Xinje XDPPro project, PLC1: XD3-48 (software 3.8.0 2025-09-09)

PROGRAM Ladder

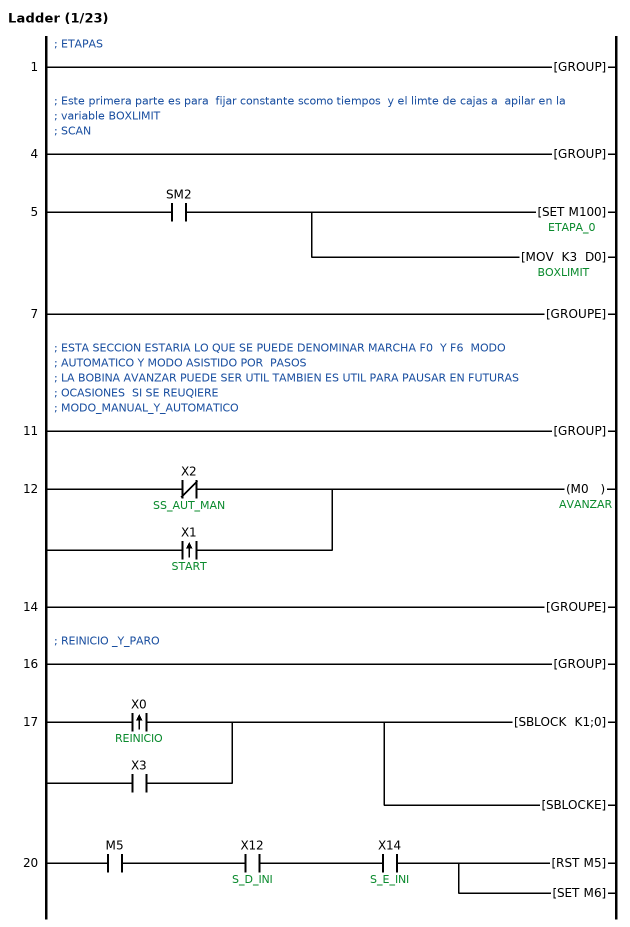
; ETAPAS
GROUP
; Este primera parte es para  fijar constante scomo tiempos  y el limte de cajas a  apilar en la variable BOXLIMIT
; SCAN
GROUP
LD     SM2
SET    M100	; ETAPA_0
MOV    K3 D0	; BOXLIMIT
GROUPE
; ESTA SECCION ESTARIA LO QUE SE PUEDE DENOMINAR MARCHA F0  Y F6  MODO AUTOMATICO Y MODO ASISTIDO POR  PASOS
; LA BOBINA AVANZAR PUEDE SER UTIL TAMBIEN ES UTIL PARA PAUSAR EN FUTURAS OCASIONES  SI SE REUQIERE
; MODO_MANUAL_Y_AUTOMATICO
GROUP
LDI    X2	; SS_AUT_MAN
ORP    X1	; START
OUT    M0	; AVANZAR
GROUPE
; REINICIO _Y_PARO
GROUP
LDP    X0	; REINICIO
OR     X3
SBLOCK K1;0
SBLOCKE
LD     M5
AND    X12	; S_D_INI
AND    X14	; S_E_INI
RST    M5
SET    M6

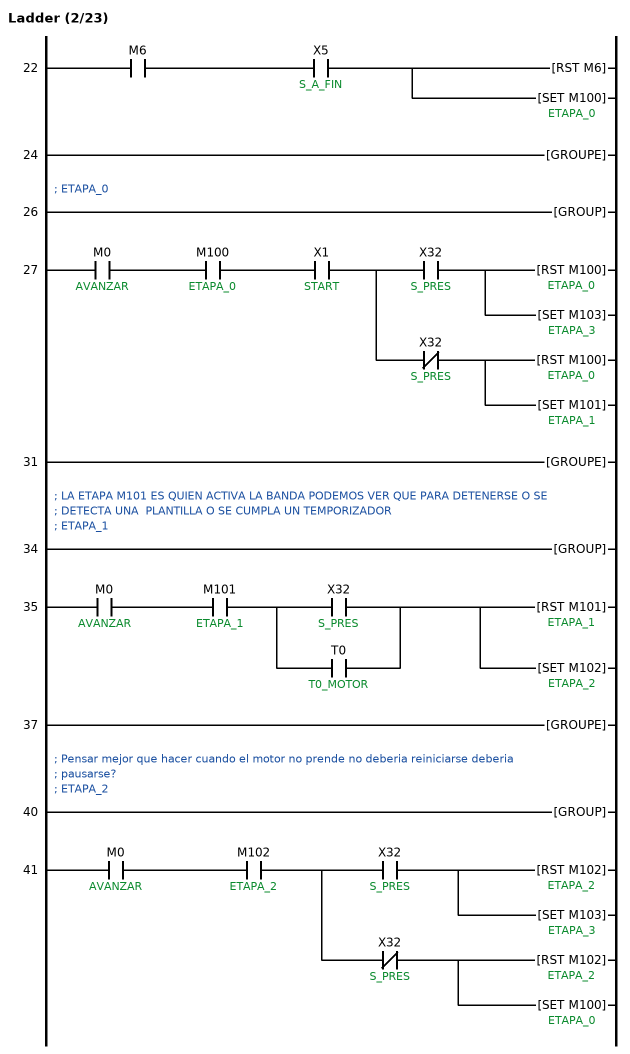
LD     M6
AND    X5	; S_A_FIN
RST    M6
SET    M100	; ETAPA_0
GROUPE
; ETAPA_0
GROUP
LD     M0	; AVANZAR
AND    M100	; ETAPA_0
AND    X1	; START
MPS
AND    X32	; S_PRES
RST    M100	; ETAPA_0
SET    M103	; ETAPA_3
MPP
ANI    X32	; S_PRES
RST    M100	; ETAPA_0
SET    M101	; ETAPA_1
GROUPE
; LA ETAPA M101 ES QUIEN ACTIVA LA BANDA PODEMOS VER QUE PARA DETENERSE O SE DETECTA UNA  PLANTILLA O SE CUMPLA UN TEMPORIZADOR 
; ETAPA_1
GROUP
LD     M0	; AVANZAR
AND    M101	; ETAPA_1
LD     X32	; S_PRES
OR     T0	; T0_MOTOR
ANB
RST    M101	; ETAPA_1
SET    M102	; ETAPA_2
GROUPE
; Pensar mejor que hacer cuando el motor no prende no deberia reiniciarse deberia pausarse?
; ETAPA_2
GROUP
LD     M0	; AVANZAR
AND    M102	; ETAPA_2
MPS
AND    X32	; S_PRES
RST    M102	; ETAPA_2
SET    M103	; ETAPA_3
MPP
ANI    X32	; S_PRES
RST    M102	; ETAPA_2
SET    M100	; ETAPA_0

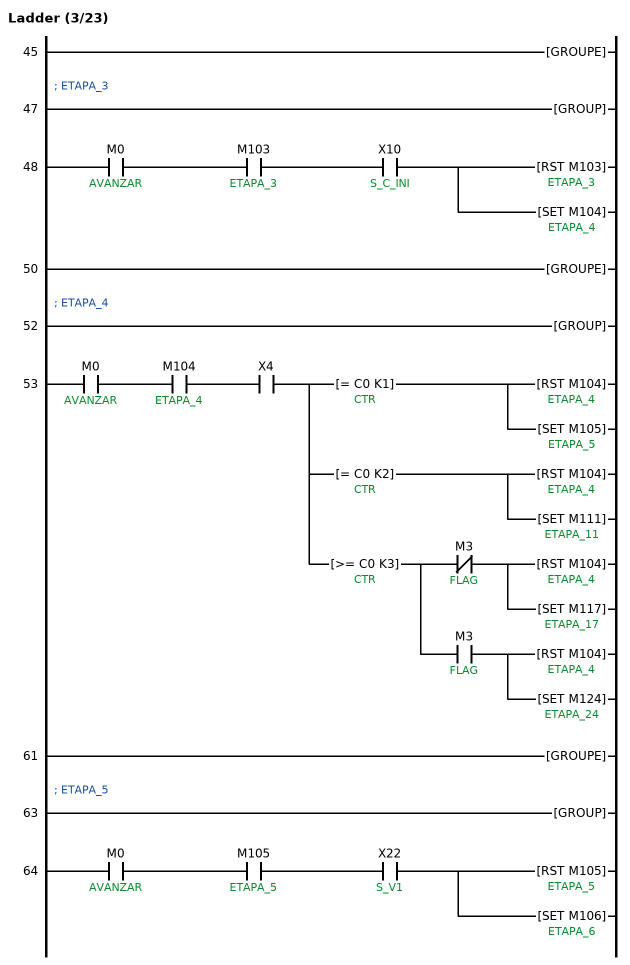
GROUPE
; ETAPA_3
GROUP
LD     M0	; AVANZAR
AND    M103	; ETAPA_3
AND    X10	; S_C_INI
RST    M103	; ETAPA_3
SET    M104	; ETAPA_4
GROUPE
; ETAPA_4
GROUP
LD     M0	; AVANZAR
AND    M104	; ETAPA_4
AND    X4
MPS
AND=   C0 K1	; CTR
RST    M104	; ETAPA_4
SET    M105	; ETAPA_5
MRD
AND=   C0 K2	; CTR
RST    M104	; ETAPA_4
SET    M111	; ETAPA_11
MPP
AND>=  C0 K3	; CTR
MPS
ANI    M3	; FLAG
RST    M104	; ETAPA_4
SET    M117	; ETAPA_17
MPP
AND    M3	; FLAG
RST    M104	; ETAPA_4
SET    M124	; ETAPA_24
GROUPE
; ETAPA_5
GROUP
LD     M0	; AVANZAR
AND    M105	; ETAPA_5
AND    X22	; S_V1
RST    M105	; ETAPA_5
SET    M106	; ETAPA_6

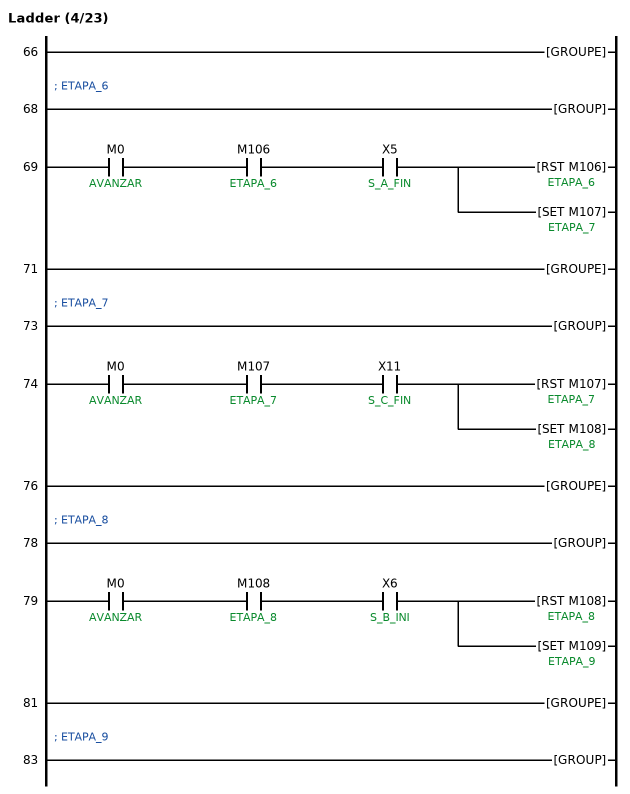
GROUPE
; ETAPA_6
GROUP
LD     M0	; AVANZAR
AND    M106	; ETAPA_6
AND    X5	; S_A_FIN
RST    M106	; ETAPA_6
SET    M107	; ETAPA_7
GROUPE
; ETAPA_7
GROUP
LD     M0	; AVANZAR
AND    M107	; ETAPA_7
AND    X11	; S_C_FIN
RST    M107	; ETAPA_7
SET    M108	; ETAPA_8
GROUPE
; ETAPA_8
GROUP
LD     M0	; AVANZAR
AND    M108	; ETAPA_8
AND    X6	; S_B_INI
RST    M108	; ETAPA_8
SET    M109	; ETAPA_9
GROUPE
; ETAPA_9
GROUP

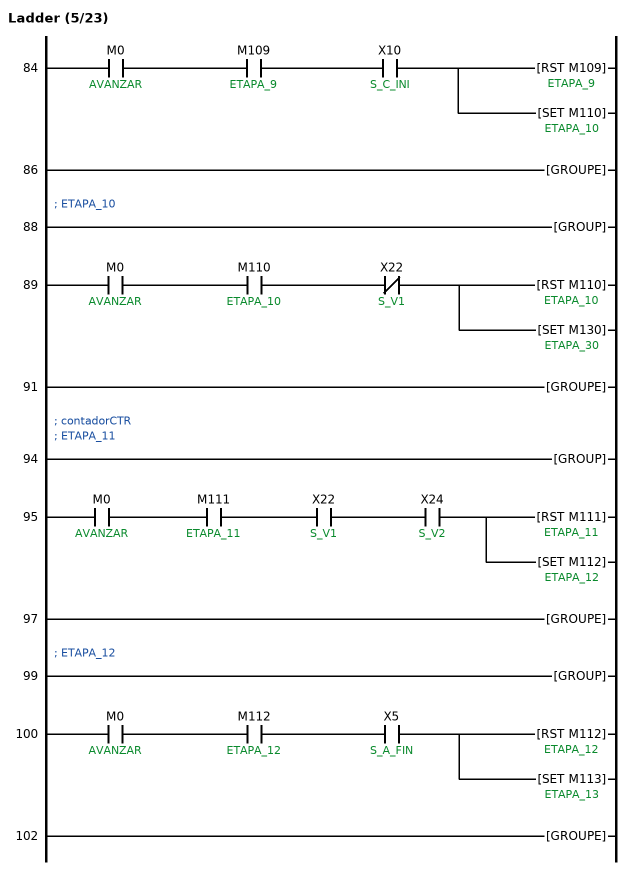
LD     M0	; AVANZAR
AND    M109	; ETAPA_9
AND    X10	; S_C_INI
RST    M109	; ETAPA_9
SET    M110	; ETAPA_10
GROUPE
; ETAPA_10
GROUP
LD     M0	; AVANZAR
AND    M110	; ETAPA_10
ANI    X22	; S_V1
RST    M110	; ETAPA_10
SET    M130	; ETAPA_30
GROUPE
; contadorCTR
; ETAPA_11
GROUP
LD     M0	; AVANZAR
AND    M111	; ETAPA_11
AND    X22	; S_V1
AND    X24	; S_V2
RST    M111	; ETAPA_11
SET    M112	; ETAPA_12
GROUPE
; ETAPA_12
GROUP
LD     M0	; AVANZAR
AND    M112	; ETAPA_12
AND    X5	; S_A_FIN
RST    M112	; ETAPA_12
SET    M113	; ETAPA_13
GROUPE

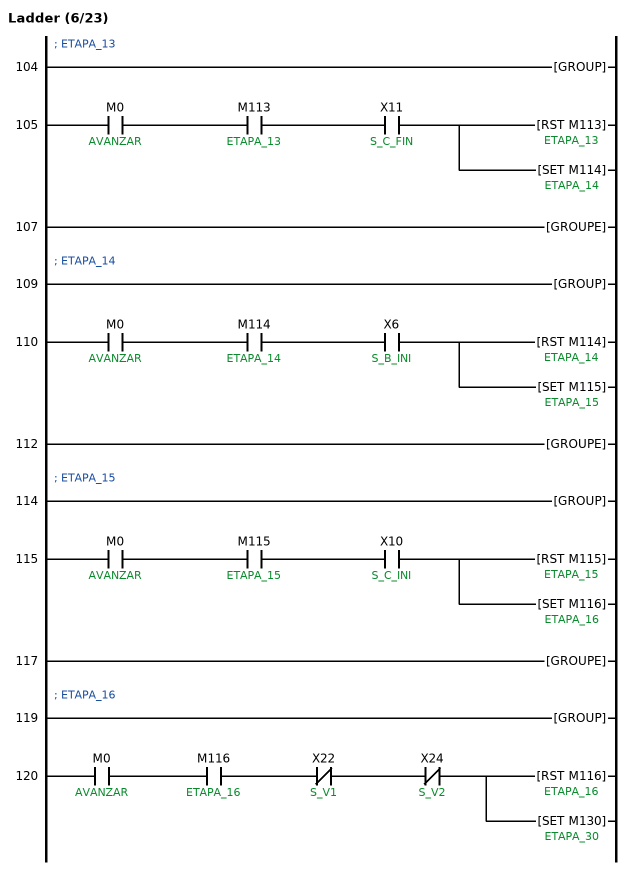
; ETAPA_13
GROUP
LD     M0	; AVANZAR
AND    M113	; ETAPA_13
AND    X11	; S_C_FIN
RST    M113	; ETAPA_13
SET    M114	; ETAPA_14
GROUPE
; ETAPA_14
GROUP
LD     M0	; AVANZAR
AND    M114	; ETAPA_14
AND    X6	; S_B_INI
RST    M114	; ETAPA_14
SET    M115	; ETAPA_15
GROUPE
; ETAPA_15
GROUP
LD     M0	; AVANZAR
AND    M115	; ETAPA_15
AND    X10	; S_C_INI
RST    M115	; ETAPA_15
SET    M116	; ETAPA_16
GROUPE
; ETAPA_16
GROUP
LD     M0	; AVANZAR
AND    M116	; ETAPA_16
ANI    X22	; S_V1
ANI    X24	; S_V2
RST    M116	; ETAPA_16
SET    M130	; ETAPA_30

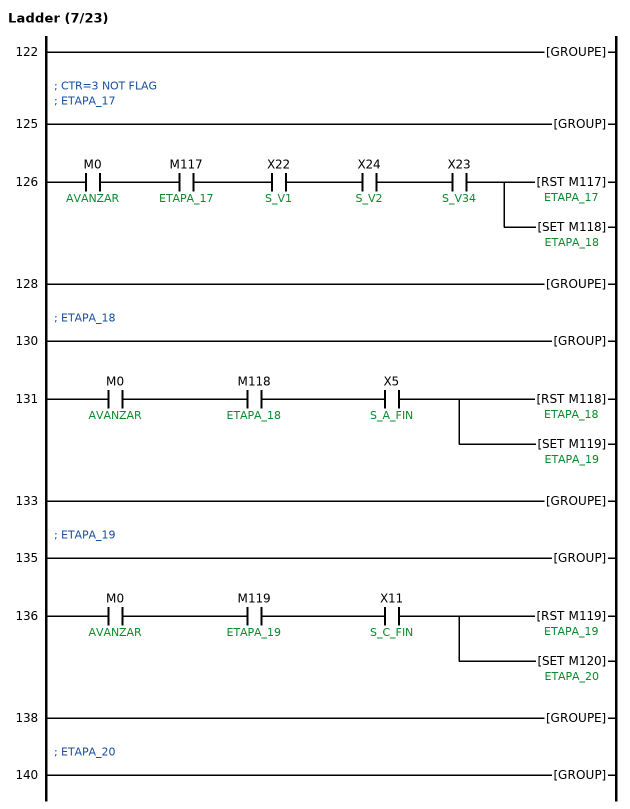
GROUPE
; CTR=3 NOT FLAG
; ETAPA_17
GROUP
LD     M0	; AVANZAR
AND    M117	; ETAPA_17
AND    X22	; S_V1
AND    X24	; S_V2
AND    X23	; S_V34
RST    M117	; ETAPA_17
SET    M118	; ETAPA_18
GROUPE
; ETAPA_18
GROUP
LD     M0	; AVANZAR
AND    M118	; ETAPA_18
AND    X5	; S_A_FIN
RST    M118	; ETAPA_18
SET    M119	; ETAPA_19
GROUPE
; ETAPA_19
GROUP
LD     M0	; AVANZAR
AND    M119	; ETAPA_19
AND    X11	; S_C_FIN
RST    M119	; ETAPA_19
SET    M120	; ETAPA_20
GROUPE
; ETAPA_20
GROUP

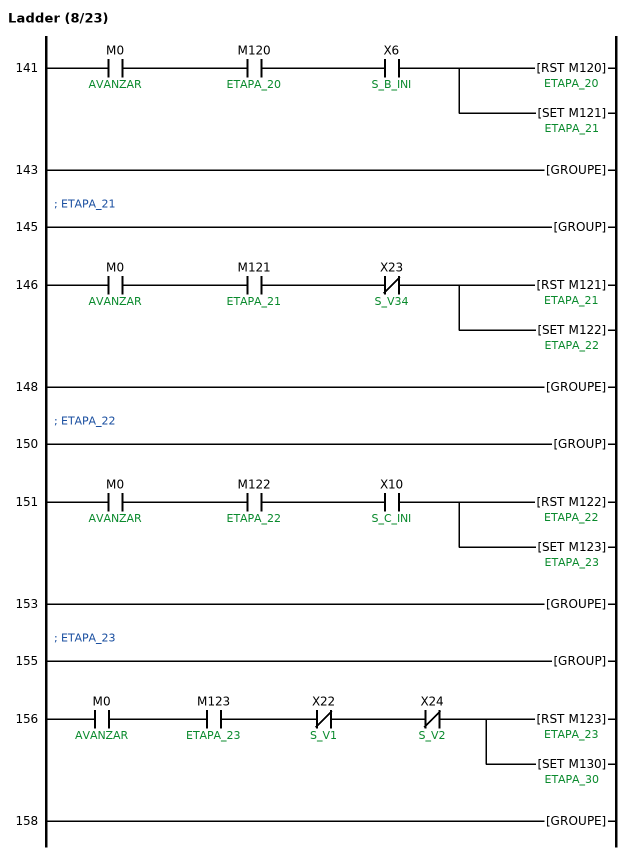
LD     M0	; AVANZAR
AND    M120	; ETAPA_20
AND    X6	; S_B_INI
RST    M120	; ETAPA_20
SET    M121	; ETAPA_21
GROUPE
; ETAPA_21
GROUP
LD     M0	; AVANZAR
AND    M121	; ETAPA_21
ANI    X23	; S_V34
RST    M121	; ETAPA_21
SET    M122	; ETAPA_22
GROUPE
; ETAPA_22
GROUP
LD     M0	; AVANZAR
AND    M122	; ETAPA_22
AND    X10	; S_C_INI
RST    M122	; ETAPA_22
SET    M123	; ETAPA_23
GROUPE
; ETAPA_23
GROUP
LD     M0	; AVANZAR
AND    M123	; ETAPA_23
ANI    X22	; S_V1
ANI    X24	; S_V2
RST    M123	; ETAPA_23
SET    M130	; ETAPA_30
GROUPE

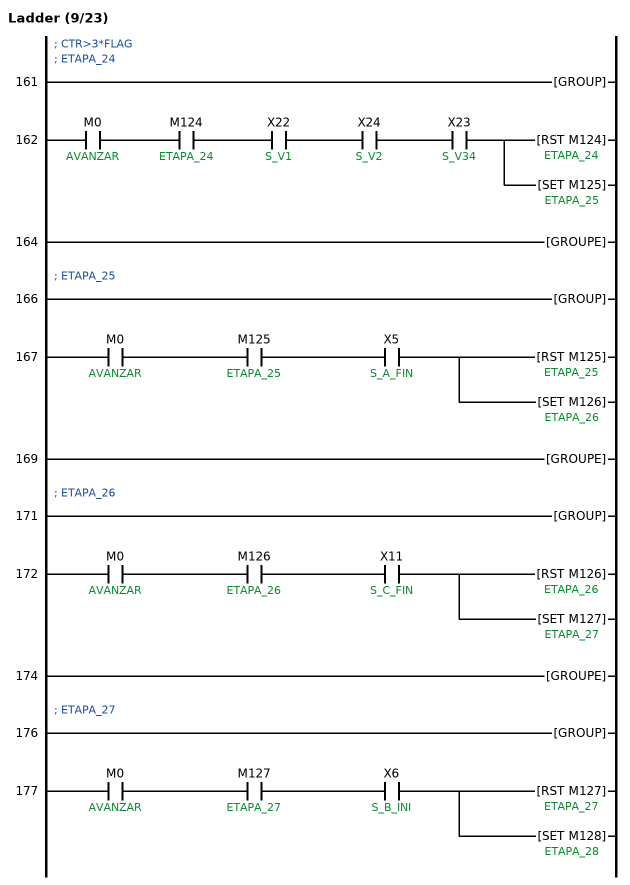
; CTR>3*FLAG
; ETAPA_24
GROUP
LD     M0	; AVANZAR
AND    M124	; ETAPA_24
AND    X22	; S_V1
AND    X24	; S_V2
AND    X23	; S_V34
RST    M124	; ETAPA_24
SET    M125	; ETAPA_25
GROUPE
; ETAPA_25
GROUP
LD     M0	; AVANZAR
AND    M125	; ETAPA_25
AND    X5	; S_A_FIN
RST    M125	; ETAPA_25
SET    M126	; ETAPA_26
GROUPE
; ETAPA_26
GROUP
LD     M0	; AVANZAR
AND    M126	; ETAPA_26
AND    X11	; S_C_FIN
RST    M126	; ETAPA_26
SET    M127	; ETAPA_27
GROUPE
; ETAPA_27
GROUP
LD     M0	; AVANZAR
AND    M127	; ETAPA_27
AND    X6	; S_B_INI
RST    M127	; ETAPA_27
SET    M128	; ETAPA_28

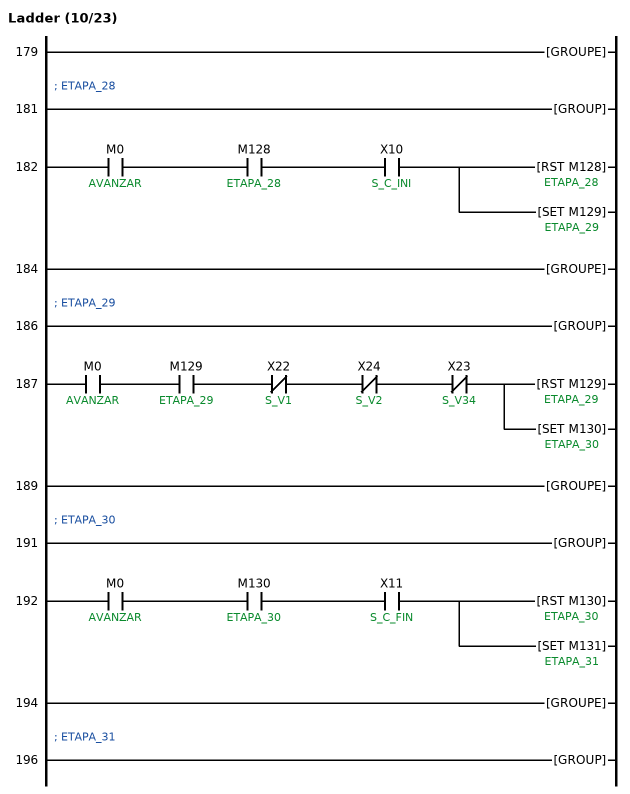
GROUPE
; ETAPA_28
GROUP
LD     M0	; AVANZAR
AND    M128	; ETAPA_28
AND    X10	; S_C_INI
RST    M128	; ETAPA_28
SET    M129	; ETAPA_29
GROUPE
; ETAPA_29
GROUP
LD     M0	; AVANZAR
AND    M129	; ETAPA_29
ANI    X22	; S_V1
ANI    X24	; S_V2
ANI    X23	; S_V34
RST    M129	; ETAPA_29
SET    M130	; ETAPA_30
GROUPE
; ETAPA_30
GROUP
LD     M0	; AVANZAR
AND    M130	; ETAPA_30
AND    X11	; S_C_FIN
RST    M130	; ETAPA_30
SET    M131	; ETAPA_31
GROUPE
; ETAPA_31
GROUP

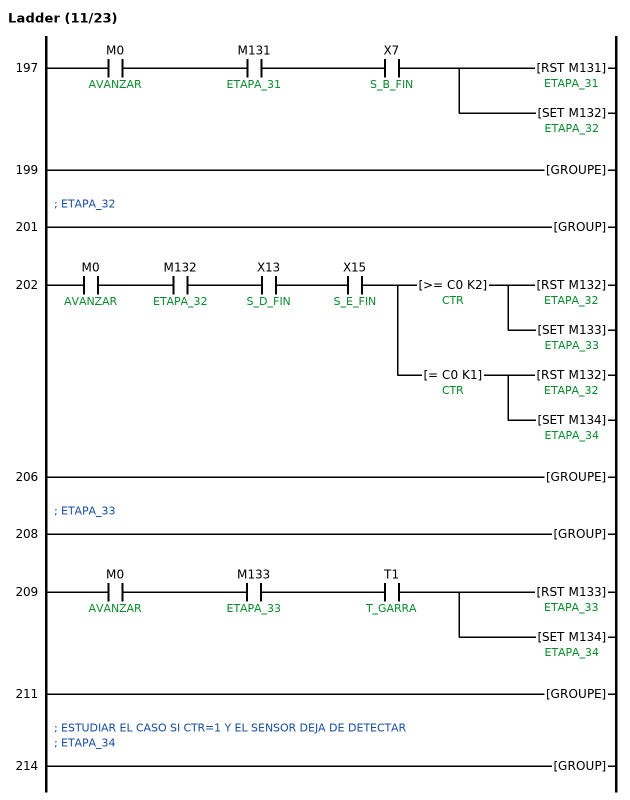
LD     M0	; AVANZAR
AND    M131	; ETAPA_31
AND    X7	; S_B_FIN
RST    M131	; ETAPA_31
SET    M132	; ETAPA_32
GROUPE
; ETAPA_32
GROUP
LD     M0	; AVANZAR
AND    M132	; ETAPA_32
AND    X13	; S_D_FIN
AND    X15	; S_E_FIN
MPS
AND>=  C0 K2	; CTR
RST    M132	; ETAPA_32
SET    M133	; ETAPA_33
MPP
AND=   C0 K1	; CTR
RST    M132	; ETAPA_32
SET    M134	; ETAPA_34
GROUPE
; ETAPA_33
GROUP
LD     M0	; AVANZAR
AND    M133	; ETAPA_33
AND    T1	; T_GARRA
RST    M133	; ETAPA_33
SET    M134	; ETAPA_34
GROUPE
; ESTUDIAR EL CASO SI CTR=1 Y EL SENSOR DEJA DE DETECTAR
; ETAPA_34
GROUP

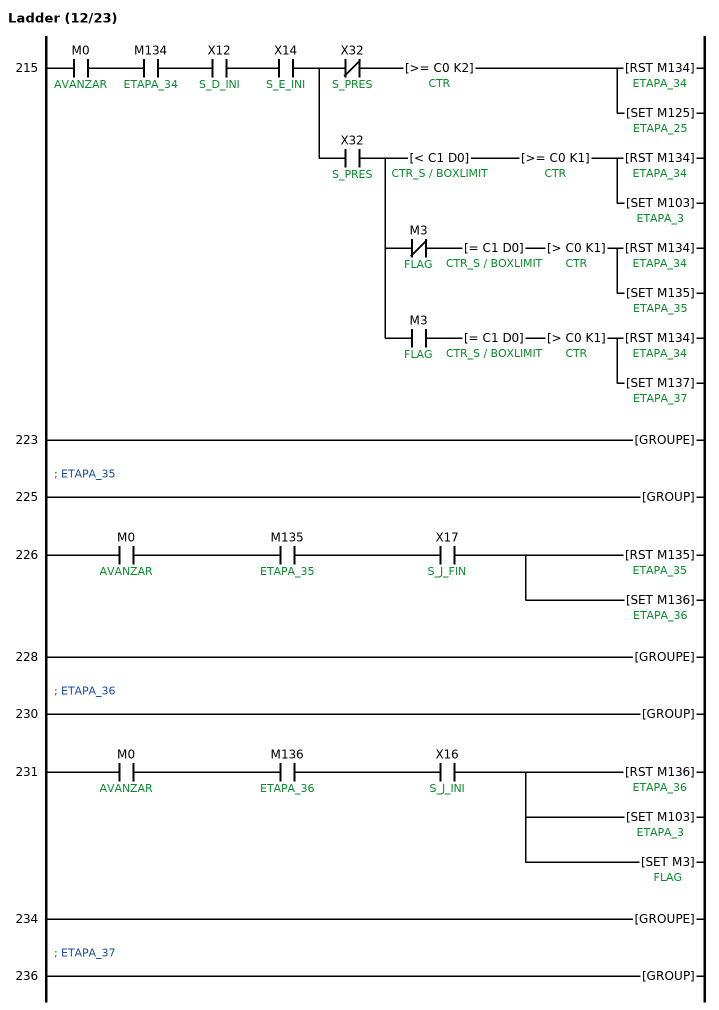
LD     M0	; AVANZAR
AND    M134	; ETAPA_34
AND    X12	; S_D_INI
AND    X14	; S_E_INI
MPS
ANI    X32	; S_PRES
AND>=  C0 K2	; CTR
RST    M134	; ETAPA_34
SET    M125	; ETAPA_25
MPP
AND    X32	; S_PRES
MPS
AND<   C1 D0	; CTR_S / BOXLIMIT
AND>=  C0 K1	; CTR
RST    M134	; ETAPA_34
SET    M103	; ETAPA_3
MRD
ANI    M3	; FLAG
AND=   C1 D0	; CTR_S / BOXLIMIT
AND>   C0 K1	; CTR
RST    M134	; ETAPA_34
SET    M135	; ETAPA_35
MPP
AND    M3	; FLAG
AND=   C1 D0	; CTR_S / BOXLIMIT
AND>   C0 K1	; CTR
RST    M134	; ETAPA_34
SET    M137	; ETAPA_37
GROUPE
; ETAPA_35
GROUP
LD     M0	; AVANZAR
AND    M135	; ETAPA_35
AND    X17	; S_J_FIN
RST    M135	; ETAPA_35
SET    M136	; ETAPA_36
GROUPE
; ETAPA_36
GROUP
LD     M0	; AVANZAR
AND    M136	; ETAPA_36
AND    X16	; S_J_INI
RST    M136	; ETAPA_36
SET    M103	; ETAPA_3
SET    M3	; FLAG
GROUPE
; ETAPA_37
GROUP

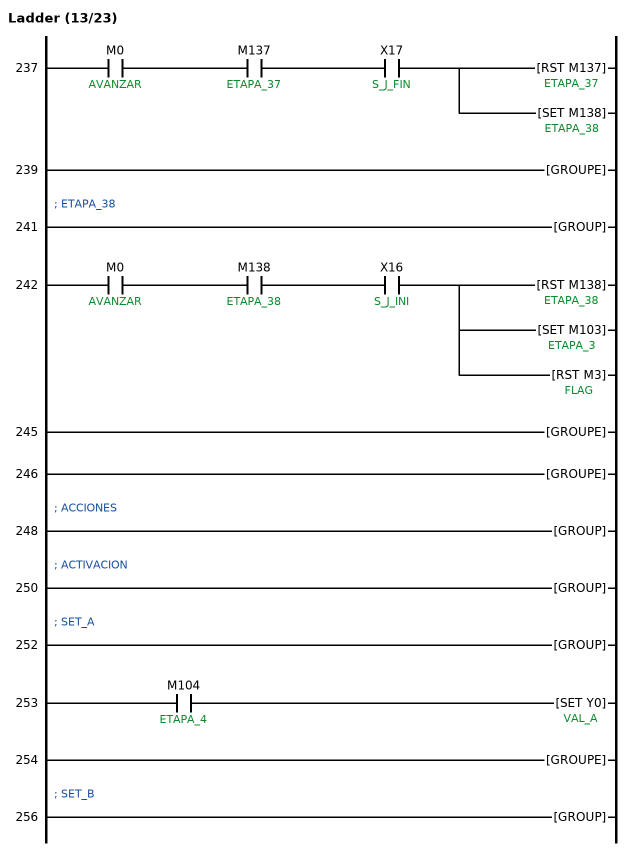
LD     M0	; AVANZAR
AND    M137	; ETAPA_37
AND    X17	; S_J_FIN
RST    M137	; ETAPA_37
SET    M138	; ETAPA_38
GROUPE
; ETAPA_38
GROUP
LD     M0	; AVANZAR
AND    M138	; ETAPA_38
AND    X16	; S_J_INI
RST    M138	; ETAPA_38
SET    M103	; ETAPA_3
RST    M3	; FLAG
GROUPE
GROUPE
; ACCIONES
GROUP
; ACTIVACION
GROUP
; SET_A
GROUP
LD     M104	; ETAPA_4
SET    Y0	; VAL_A
GROUPE
; SET_B
GROUP

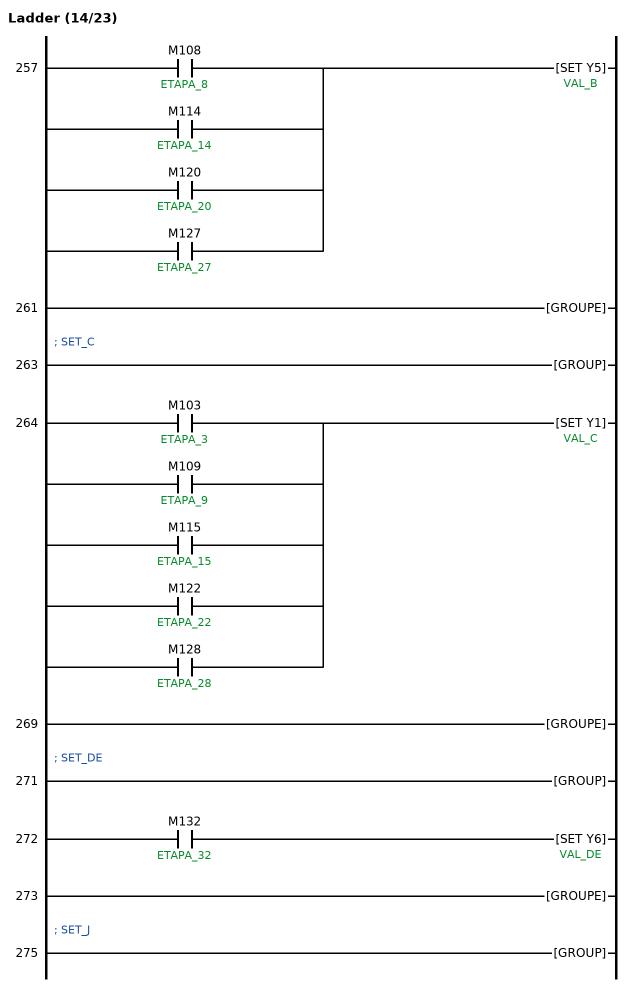
LD     M108	; ETAPA_8
OR     M114	; ETAPA_14
OR     M120	; ETAPA_20
OR     M127	; ETAPA_27
SET    Y5	; VAL_B
GROUPE
; SET_C
GROUP
LD     M103	; ETAPA_3
OR     M109	; ETAPA_9
OR     M115	; ETAPA_15
OR     M122	; ETAPA_22
OR     M128	; ETAPA_28
SET    Y1	; VAL_C
GROUPE
; SET_DE
GROUP
LD     M132	; ETAPA_32
SET    Y6	; VAL_DE
GROUPE
; SET_J
GROUP

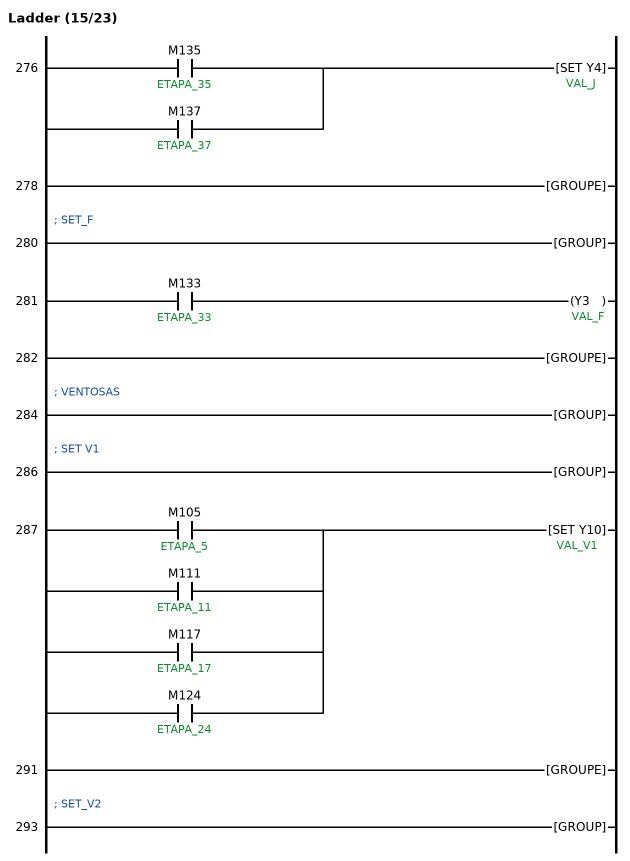
LD     M135	; ETAPA_35
OR     M137	; ETAPA_37
SET    Y4	; VAL_J
GROUPE
; SET_F
GROUP
LD     M133	; ETAPA_33
OUT    Y3	; VAL_F
GROUPE
; VENTOSAS
GROUP
; SET V1
GROUP
LD     M105	; ETAPA_5
OR     M111	; ETAPA_11
OR     M117	; ETAPA_17
OR     M124	; ETAPA_24
SET    Y10	; VAL_V1
GROUPE
; SET_V2
GROUP

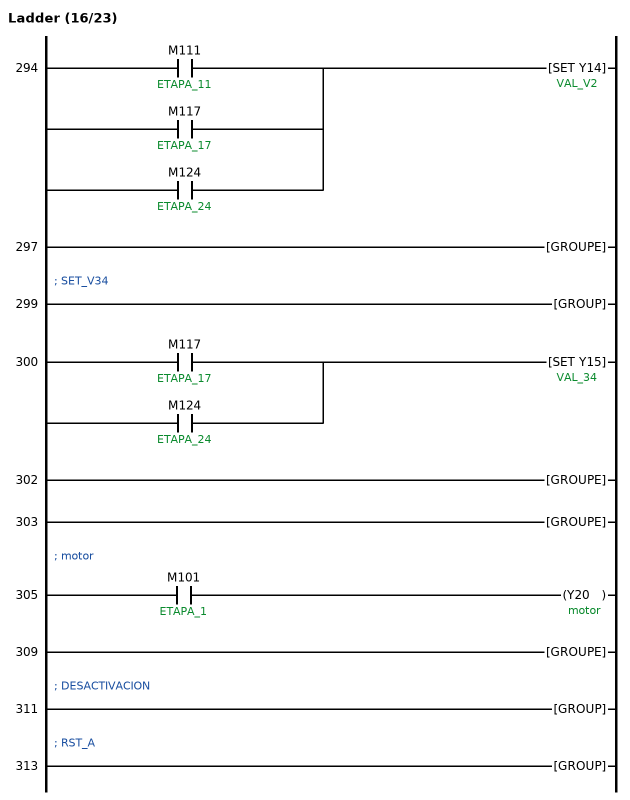
LD     M111	; ETAPA_11
OR     M117	; ETAPA_17
OR     M124	; ETAPA_24
SET    Y14	; VAL_V2
GROUPE
; SET_V34
GROUP
LD     M117	; ETAPA_17
OR     M124	; ETAPA_24
SET    Y15	; VAL_34
GROUPE
GROUPE
; motor
LD     M101	; ETAPA_1
OUT    Y20	; motor
GROUPE
; DESACTIVACION
GROUP
; RST_A
GROUP

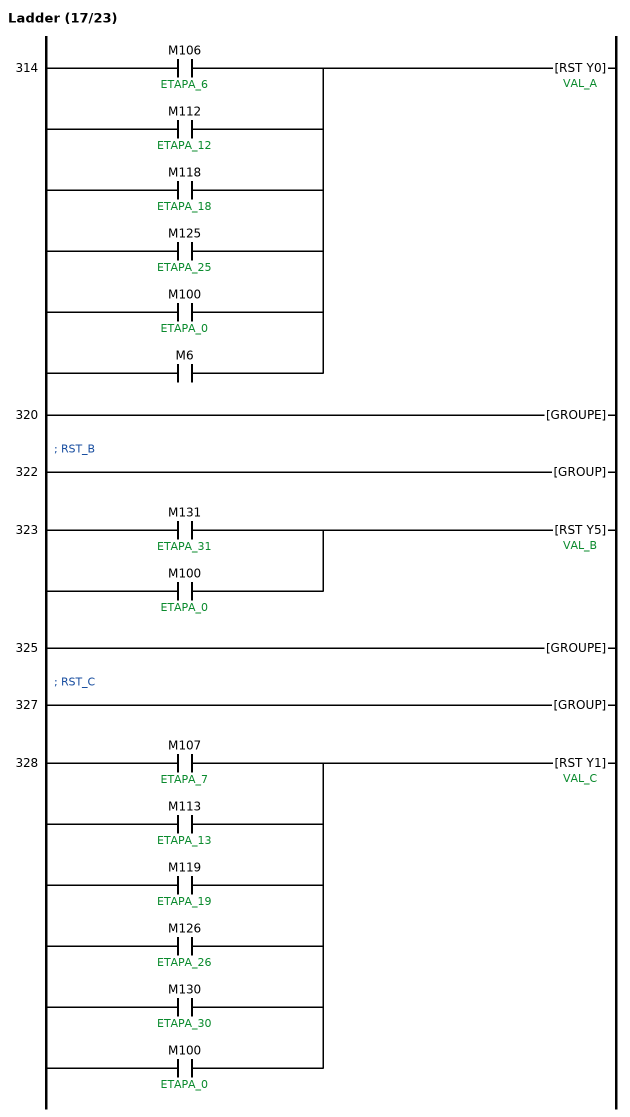
LD     M106	; ETAPA_6
OR     M112	; ETAPA_12
OR     M118	; ETAPA_18
OR     M125	; ETAPA_25
OR     M100	; ETAPA_0
OR     M6
RST    Y0	; VAL_A
GROUPE
; RST_B
GROUP
LD     M131	; ETAPA_31
OR     M100	; ETAPA_0
RST    Y5	; VAL_B
GROUPE
; RST_C
GROUP
LD     M107	; ETAPA_7
OR     M113	; ETAPA_13
OR     M119	; ETAPA_19
OR     M126	; ETAPA_26
OR     M130	; ETAPA_30
OR     M100	; ETAPA_0
RST    Y1	; VAL_C

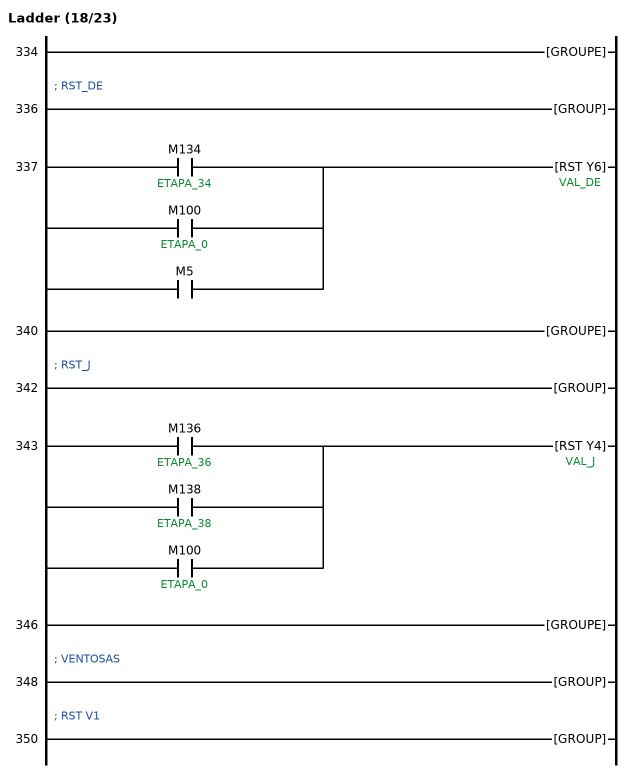
GROUPE
; RST_DE
GROUP
LD     M134	; ETAPA_34
OR     M100	; ETAPA_0
OR     M5
RST    Y6	; VAL_DE
GROUPE
; RST_J
GROUP
LD     M136	; ETAPA_36
OR     M138	; ETAPA_38
OR     M100	; ETAPA_0
RST    Y4	; VAL_J
GROUPE
; VENTOSAS
GROUP
; RST V1
GROUP

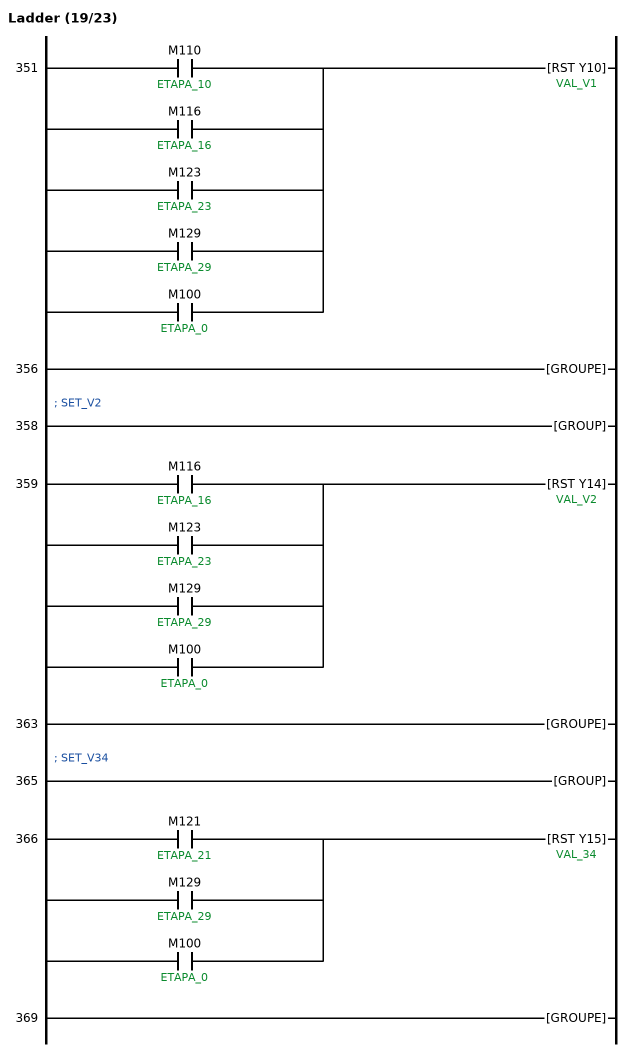
LD     M110	; ETAPA_10
OR     M116	; ETAPA_16
OR     M123	; ETAPA_23
OR     M129	; ETAPA_29
OR     M100	; ETAPA_0
RST    Y10	; VAL_V1
GROUPE
; SET_V2
GROUP
LD     M116	; ETAPA_16
OR     M123	; ETAPA_23
OR     M129	; ETAPA_29
OR     M100	; ETAPA_0
RST    Y14	; VAL_V2
GROUPE
; SET_V34
GROUP
LD     M121	; ETAPA_21
OR     M129	; ETAPA_29
OR     M100	; ETAPA_0
RST    Y15	; VAL_34
GROUPE

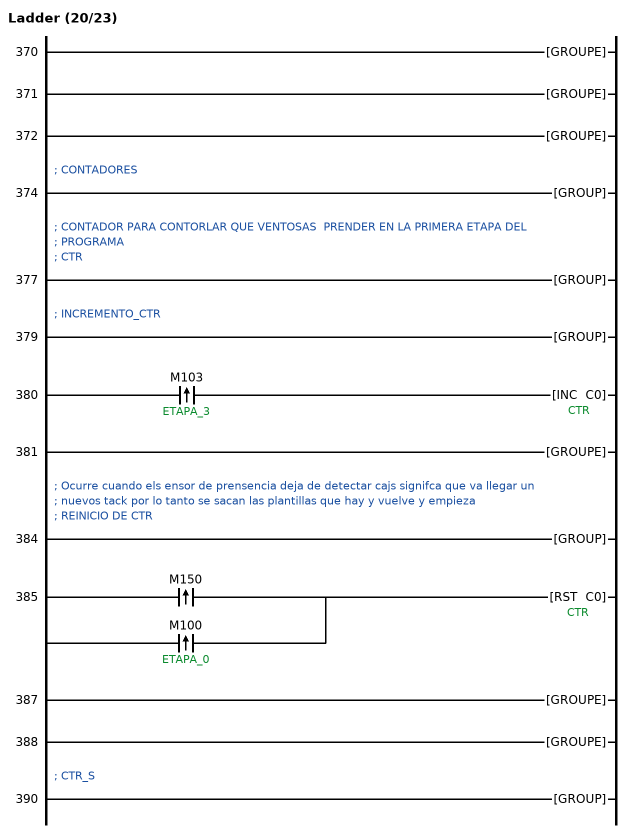
GROUPE
GROUPE
GROUPE
; CONTADORES
GROUP
; CONTADOR PARA CONTORLAR QUE VENTOSAS  PRENDER EN LA PRIMERA ETAPA DEL PROGRAMA
; CTR
GROUP
; INCREMENTO_CTR
GROUP
LDP    M103	; ETAPA_3
INC    C0	; CTR
GROUPE
; Ocurre cuando els ensor de prensencia deja de detectar cajs signifca que va llegar un nuevos tack por lo tanto se sacan las plantillas que hay y vuelve y empieza
; REINICIO DE CTR
GROUP
LDP    M150
ORP    M100	; ETAPA_0
RST    C0	; CTR
GROUPE
GROUPE
; CTR_S
GROUP

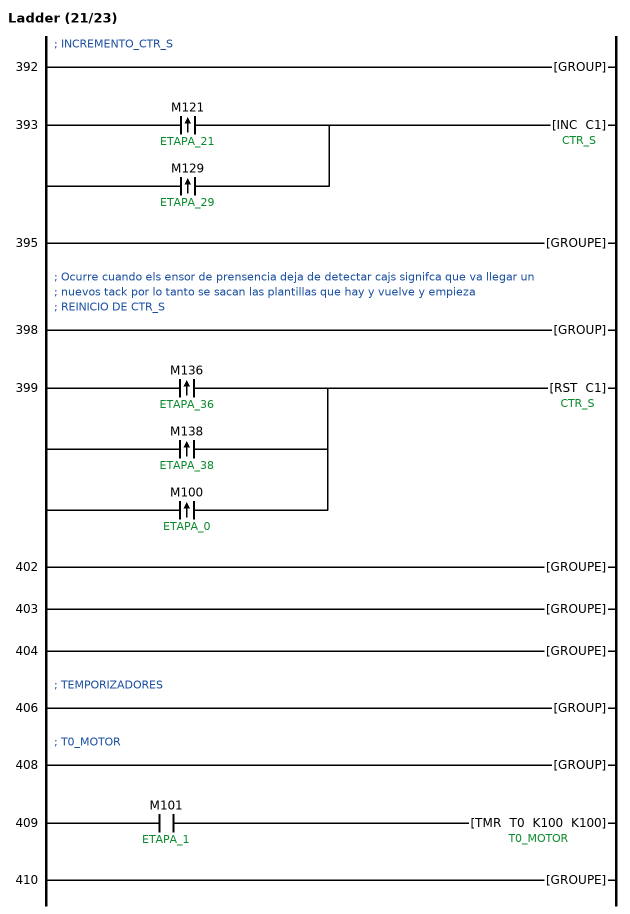
; INCREMENTO_CTR_S
GROUP
LDP    M121	; ETAPA_21
ORP    M129	; ETAPA_29
INC    C1	; CTR_S
GROUPE
; Ocurre cuando els ensor de prensencia deja de detectar cajs signifca que va llegar un nuevos tack por lo tanto se sacan las plantillas que hay y vuelve y empieza
; REINICIO DE CTR_S
GROUP
LDP    M136	; ETAPA_36
ORP    M138	; ETAPA_38
ORP    M100	; ETAPA_0
RST    C1	; CTR_S
GROUPE
GROUPE
GROUPE
; TEMPORIZADORES
GROUP
; T0_MOTOR
GROUP
LD     M101	; ETAPA_1
TMR    T0 K100 K100	; T0_MOTOR
GROUPE

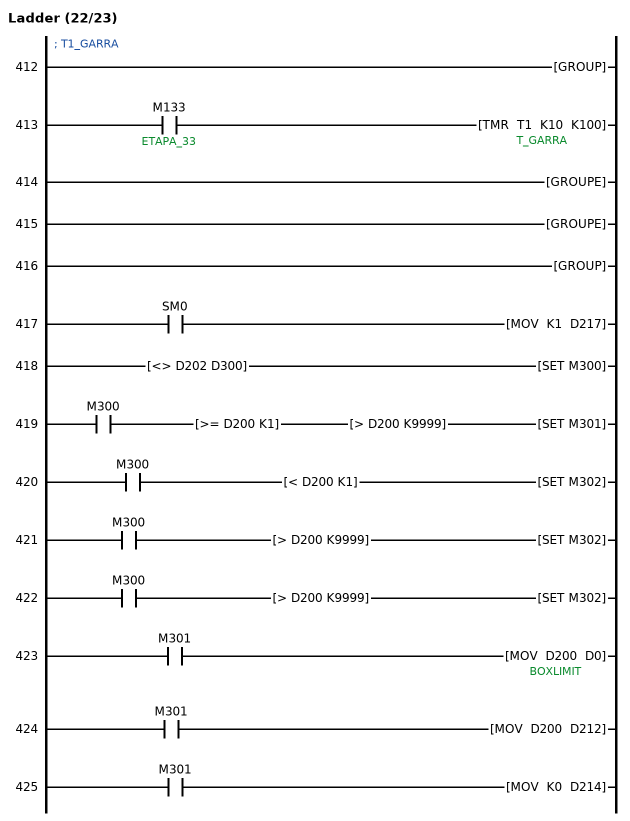
; T1_GARRA
GROUP
LD     M133	; ETAPA_33
TMR    T1 K10 K100	; T_GARRA
GROUPE
GROUPE
GROUP
LD     SM0
MOV    K1 D217
LD<>   D202 D300
SET    M300
LD     M300
AND>=  D200 K1
AND>   D200 K9999
SET    M301
LD     M300
AND<   D200 K1
SET    M302
LD     M300
AND>   D200 K9999
SET    M302
LD     M300
AND>   D200 K9999
SET    M302
LD     M301
MOV    D200 D0	; BOXLIMIT
LD     M301
MOV    D200 D212
LD     M301
MOV    K0 D214

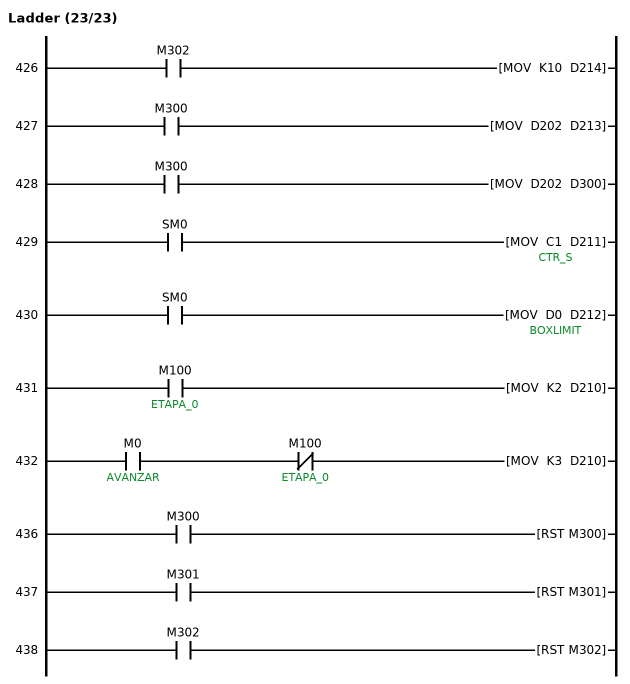
LD     M302
MOV    K10 D214
LD     M300
MOV    D202 D213
LD     M300
MOV    D202 D300
LD     SM0
MOV    C1 D211	; CTR_S
LD     SM0
MOV    D0 D212	; BOXLIMIT
LD     M100	; ETAPA_0
MOV    K2 D210
LD     M0	; AVANZAR
ANI    M100	; ETAPA_0
MOV    K3 D210
LD     M300
RST    M300
LD     M301
RST    M301
LD     M302
RST    M302

SBLOCK K1	; Sequence Block1
  ; Instruction List
  LD<> DM101 K0
  OR<> DM116 K0
  OR<> DM132 K0
  OR<> DM148 K0
  ZRST M101 M156
  SET M5